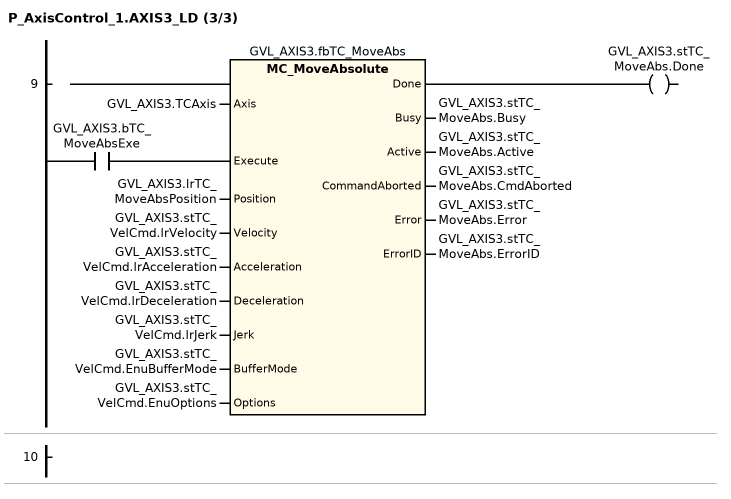
// NETWORK 9
GVL_AXIS3.fbTC_MoveAbs(
    Axis := GVL_AXIS3.TCAxis,
    Execute := GVL_AXIS3.bTC_MoveAbsExe,
    Position := GVL_AXIS3.lrTC_MoveAbsPosition,
    Velocity := GVL_AXIS3.stTC_VelCmd.lrVelocity,
    Acceleration := GVL_AXIS3.stTC_VelCmd.lrAcceleration,
    Deceleration := GVL_AXIS3.stTC_VelCmd.lrDeceleration,
    Jerk := GVL_AXIS3.stTC_VelCmd.lrJerk,
    BufferMode := GVL_AXIS3.stTC_VelCmd.EnuBufferMode,
    Options := GVL_AXIS3.stTC_VelCmd.EnuOptions,
    Busy => GVL_AXIS3.stTC_MoveAbs.Busy,
    Active => GVL_AXIS3.stTC_MoveAbs.Active,
    CommandAborted => GVL_AXIS3.stTC_MoveAbs.CmdAborted,
    Error => GVL_AXIS3.stTC_MoveAbs.Error,
    ErrorID => GVL_AXIS3.stTC_MoveAbs.ErrorID); // MC_MoveAbsolute
GVL_AXIS3.stTC_MoveAbs.Done := GVL_AXIS3.fbTC_MoveAbs.Done;

// NETWORK 10
END_METHOD

METHOD AXIS4_LD : BOOL
VAR_INPUT
END_VAR
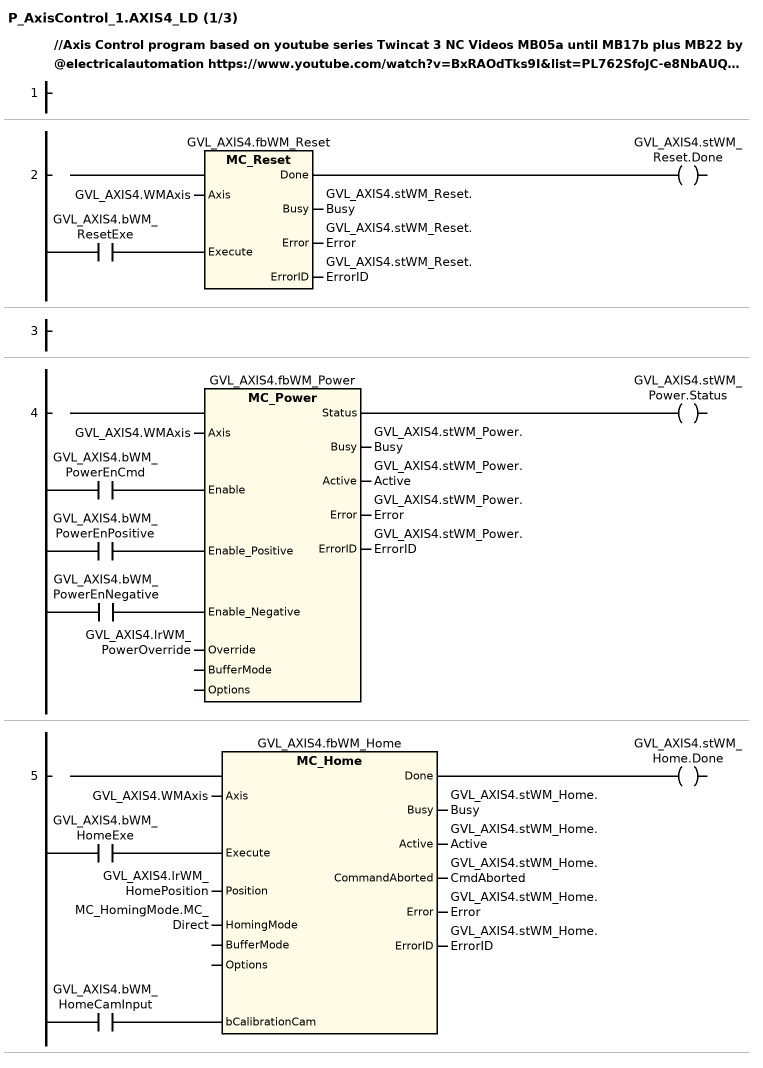
// NETWORK 1: //Axis Control program based on youtube series Twincat 3 NC Videos MB05a until MB17b plus MB22 by @electricalautomation https://www.youtube.com/watch?v=BxRAOdTks9I&list=PL762SfoJC-e8NbAUQ-H7a_TOdqrlBPCw4&index=25

// NETWORK 2
GVL_AXIS4.fbWM_Reset(
    Axis := GVL_AXIS4.WMAxis,
    Execute := GVL_AXIS4.bWM_ResetExe,
    Busy => GVL_AXIS4.stWM_Reset.Busy,
    Error => GVL_AXIS4.stWM_Reset.Error,
    ErrorID => GVL_AXIS4.stWM_Reset.ErrorID); // MC_Reset
GVL_AXIS4.stWM_Reset.Done := GVL_AXIS4.fbWM_Reset.Done;

// NETWORK 3

// NETWORK 4
GVL_AXIS4.fbWM_Power(
    Axis := GVL_AXIS4.WMAxis,
    Enable := GVL_AXIS4.bWM_PowerEnCmd,
    Enable_Positive := GVL_AXIS4.bWM_PowerEnPositive,
    Enable_Negative := GVL_AXIS4.bWM_PowerEnNegative,
    Override := GVL_AXIS4.lrWM_PowerOverride,
    Busy => GVL_AXIS4.stWM_Power.Busy,
    Active => GVL_AXIS4.stWM_Power.Active,
    Error => GVL_AXIS4.stWM_Power.Error,
    ErrorID => GVL_AXIS4.stWM_Power.ErrorID); // MC_Power
GVL_AXIS4.stWM_Power.Status := GVL_AXIS4.fbWM_Power.Status;

// NETWORK 5
GVL_AXIS4.fbWM_Home(
    Axis := GVL_AXIS4.WMAxis,
    Execute := GVL_AXIS4.bWM_HomeExe,
    Position := GVL_AXIS4.lrWM_HomePosition,
    HomingMode := MC_HomingMode.MC_Direct,
    bCalibrationCam := GVL_AXIS4.bWM_HomeCamInput,
    Busy => GVL_AXIS4.stWM_Home.Busy,
    Active => GVL_AXIS4.stWM_Home.Active,
    CommandAborted => GVL_AXIS4.stWM_Home.CmdAborted,
    Error => GVL_AXIS4.stWM_Home.Error,
    ErrorID => GVL_AXIS4.stWM_Home.ErrorID); // MC_Home
GVL_AXIS4.stWM_Home.Done := GVL_AXIS4.fbWM_Home.Done;

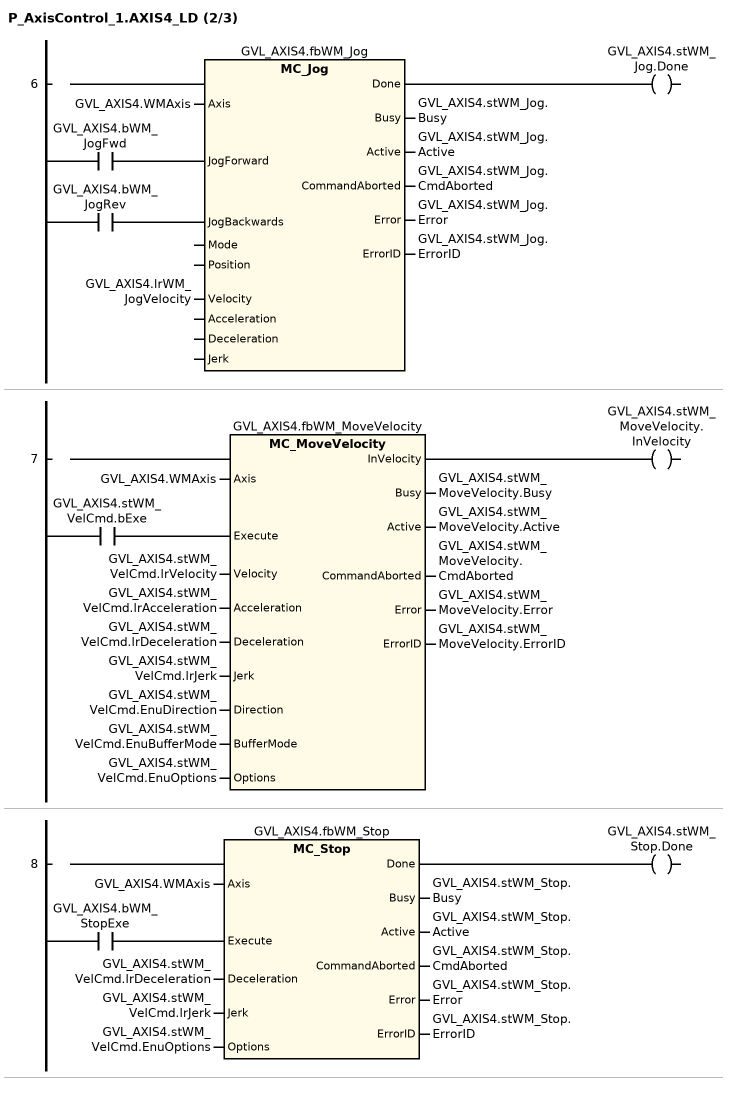
// NETWORK 6
GVL_AXIS4.fbWM_Jog(
    Axis := GVL_AXIS4.WMAxis,
    JogForward := GVL_AXIS4.bWM_JogFwd,
    JogBackwards := GVL_AXIS4.bWM_JogRev,
    Velocity := GVL_AXIS4.lrWM_JogVelocity,
    Busy => GVL_AXIS4.stWM_Jog.Busy,
    Active => GVL_AXIS4.stWM_Jog.Active,
    CommandAborted => GVL_AXIS4.stWM_Jog.CmdAborted,
    Error => GVL_AXIS4.stWM_Jog.Error,
    ErrorID => GVL_AXIS4.stWM_Jog.ErrorID); // MC_Jog
GVL_AXIS4.stWM_Jog.Done := GVL_AXIS4.fbWM_Jog.Done;

// NETWORK 7
GVL_AXIS4.fbWM_MoveVelocity(
    Axis := GVL_AXIS4.WMAxis,
    Execute := GVL_AXIS4.stWM_VelCmd.bExe,
    Velocity := GVL_AXIS4.stWM_VelCmd.lrVelocity,
    Acceleration := GVL_AXIS4.stWM_VelCmd.lrAcceleration,
    Deceleration := GVL_AXIS4.stWM_VelCmd.lrDeceleration,
    Jerk := GVL_AXIS4.stWM_VelCmd.lrJerk,
    Direction := GVL_AXIS4.stWM_VelCmd.EnuDirection,
    BufferMode := GVL_AXIS4.stWM_VelCmd.EnuBufferMode,
    Options := GVL_AXIS4.stWM_VelCmd.EnuOptions,
    Busy => GVL_AXIS4.stWM_MoveVelocity.Busy,
    Active => GVL_AXIS4.stWM_MoveVelocity.Active,
    CommandAborted => GVL_AXIS4.stWM_MoveVelocity.CmdAborted,
    Error => GVL_AXIS4.stWM_MoveVelocity.Error,
    ErrorID => GVL_AXIS4.stWM_MoveVelocity.ErrorID); // MC_MoveVelocity
GVL_AXIS4.stWM_MoveVelocity.InVelocity := GVL_AXIS4.fbWM_MoveVelocity.InVelocity;

// NETWORK 8
GVL_AXIS4.fbWM_Stop(
    Axis := GVL_AXIS4.WMAxis,
    Execute := GVL_AXIS4.bWM_StopExe,
    Deceleration := GVL_AXIS4.stWM_VelCmd.lrDeceleration,
    Jerk := GVL_AXIS4.stWM_VelCmd.lrJerk,
    Options := GVL_AXIS4.stWM_VelCmd.EnuOptions,
    Busy => GVL_AXIS4.stWM_Stop.Busy,
    Active => GVL_AXIS4.stWM_Stop.Active,
    CommandAborted => GVL_AXIS4.stWM_Stop.CmdAborted,
    Error => GVL_AXIS4.stWM_Stop.Error,
    ErrorID => GVL_AXIS4.stWM_Stop.ErrorID); // MC_Stop
GVL_AXIS4.stWM_Stop.Done := GVL_AXIS4.fbWM_Stop.Done;

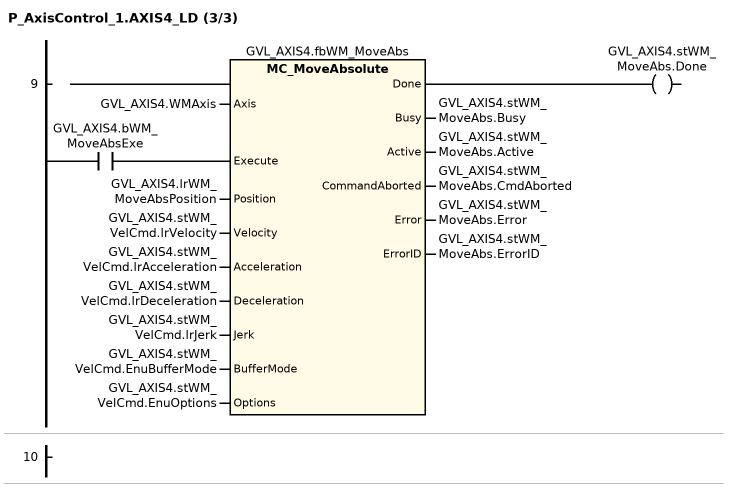
// NETWORK 9
GVL_AXIS4.fbWM_MoveAbs(
    Axis := GVL_AXIS4.WMAxis,
    Execute := GVL_AXIS4.bWM_MoveAbsExe,
    Position := GVL_AXIS4.lrWM_MoveAbsPosition,
    Velocity := GVL_AXIS4.stWM_VelCmd.lrVelocity,
    Acceleration := GVL_AXIS4.stWM_VelCmd.lrAcceleration,
    Deceleration := GVL_AXIS4.stWM_VelCmd.lrDeceleration,
    Jerk := GVL_AXIS4.stWM_VelCmd.lrJerk,
    BufferMode := GVL_AXIS4.stWM_VelCmd.EnuBufferMode,
    Options := GVL_AXIS4.stWM_VelCmd.EnuOptions,
    Busy => GVL_AXIS4.stWM_MoveAbs.Busy,
    Active => GVL_AXIS4.stWM_MoveAbs.Active,
    CommandAborted => GVL_AXIS4.stWM_MoveAbs.CmdAborted,
    Error => GVL_AXIS4.stWM_MoveAbs.Error,
    ErrorID => GVL_AXIS4.stWM_MoveAbs.ErrorID); // MC_MoveAbsolute
GVL_AXIS4.stWM_MoveAbs.Done := GVL_AXIS4.fbWM_MoveAbs.Done;

// NETWORK 10
END_METHOD

METHOD Manual_mode : BOOL
VAR_INPUT
END_VAR
AXIS1_LD();

GVL_AXIS1.bBC_ResetExe := G_Inputs.bJoystickLeftEnable;

//GVL_AXIS1.EnuMoveVelDirection := G_Sensors.MCDirectionAxis1;

GVL_AXIS1.bBC_PowerEnCmd := G_Inputs.bManualModeSelector;
GVL_AXIS1.bBC_PowerEnNegative := G_Inputs.bManualModeSelector;
GVL_AXIS1.bBC_PowerEnPositive := G_Inputs.bManualModeSelector;

IF G_Sensors.fJoystickLeftNormalizedX  > 0.01 AND G_Inputs.bJoystickLeftEnable THEN
	GVL_AXIS1.lrBC_PowerOverride := ABS(G_Sensors.fJoystickLeftNormalizedX) * 100;
	GVL_AXIS1.stBC_VelCmd.EnuDirection := MC_Positive_Direction;
	GVL_AXIS1.stBC_VelCmd.bExe := TRUE;
ELSIF G_Sensors.fJoystickLeftNormalizedX < 0.01 AND G_Inputs.bJoystickLeftEnable THEN
	GVL_AXIS1.lrBC_PowerOverride := ABS(G_Sensors.fJoystickLeftNormalizedX) * 100;
	GVL_AXIS1.stBC_VelCmd.EnuDirection := MC_Negative_Direction;
	GVL_AXIS1.stBC_VelCmd.bExe := TRUE;
END_IF
END_METHOD

END_PROGRAM

// ---- INPUTS/P_Inputs.TcPOU
PROGRAM P_Inputs
VAR
	fbJoystickLeftVert 					: FB_JoystickInputScaling;
	fbJoystickLeftHor 					: FB_JoystickInputScaling;
	
	fbJoystickRightVert 				: FB_JoystickInputScaling;
	fbJoystickRightHor 					: FB_JoystickInputScaling;
	
	bEnableJoystick : BOOL;
		
END_VAR

bEnableJoystick := NOT(P_StablePlatform.bManualMode);

fbJoystickLeftVert(
	bEnable := bEnableJoystick,
	nRawInput := G_Inputs.stJoyLY.nValue,
	stJoystickInputScaling := G_ScalingParameters.stParam.stJoystickInputScalingLeftY,
	fNormalizedOutput => G_Sensors.fJoystickLeftNormalizedY
);

IF G_Sensors.fJoystickLeftNormalizedY < 0 THEN
	G_Sensors.MCDirectionAxis3 := MC_Negative_Direction;
ELSIF G_Sensors.fJoystickLeftNormalizedY > 0 THEN
	G_Sensors.MCDirectionAxis3 := MC_Positive_Direction;	
END_IF

fbJoystickLeftHor(
	bEnable := bEnableJoystick,
	nRawInput := G_Inputs.stJoyLX.nValue,
	stJoystickInputScaling := G_ScalingParameters.stParam.stJoystickInputScalingLeftX,
	fNormalizedOutput => G_Sensors.fJoystickLeftNormalizedX
);

IF G_Sensors.fJoystickLeftNormalizedX < 0 THEN
	G_Sensors.MCDirectionAxis1 := MC_Positive_Direction;
ELSIF G_Sensors.fJoystickLeftNormalizedX > 0 THEN
	G_Sensors.MCDirectionAxis1 := MC_Negative_Direction;	
END_IF


fbJoystickRightVert(
	bEnable := bEnableJoystick,
	nRawInput := G_Inputs.stJoyRY.nValue,
	stJoystickInputScaling := G_ScalingParameters.stParam.stJoystickInputScalingRightY,
	fNormalizedOutput => G_Sensors.fJoystickRightNormalizedY
);

IF G_Sensors.fJoystickRightNormalizedY < 0 THEN
	G_Sensors.MCDirectionAxis4 := MC_Negative_Direction;
ELSIF G_Sensors.fJoystickRightNormalizedY > 0 THEN
	G_Sensors.MCDirectionAxis4 := MC_Positive_Direction;	
END_IF



fbJoystickRightHor(
	bEnable := bEnableJoystick,
	nRawInput := G_Inputs.stJoyRX.nValue,
	stJoystickInputScaling := G_ScalingParameters.stParam.stJoystickInputScalingRightX,
	fNormalizedOutput => G_Sensors.fJoystickRightNormalizedX
);

IF G_Sensors.fJoystickRightNormalizedX < 0 THEN
	G_Sensors.MCDirectionAxis2 := MC_Positive_Direction;
ELSIF G_Sensors.fJoystickRightNormalizedX > 0 THEN
	G_Sensors.MCDirectionAxis2 := MC_Negative_Direction;	
END_IF

END_PROGRAM

// ---- StablePlatform/P_StablePlatform.TcPOU
PROGRAM P_StablePlatform
VAR
	fbpA 		: FB_AnalogInputScaling;
	fbpB 		: FB_AnalogInputScaling;
	fbpS 	 	: FB_AnalogInputScaling;
	fSVFeedback : FB_AnalogInputScaling;
	fbPistonPos	: FB_AnalogInputScaling_1;
	fbPistonVel	: FB_AnalogInputScaling_1;
	fbJoystick  : FB_JoystickInputScaling;
	fbSVOutput 	: FB_ValveOutput;
	bManualMode : BOOL;
END_VAR

// Inputs
fbpA(
	nRawInput := G_StablePlatformIO.npA,
	stAnalogInputScaling := G_StablePlatformParameters.stPressureSensorScaling400bar,
	fOutput => G_StablePlatformScaledIO.bpA
);

fbpB(
	nRawInput := G_StablePlatformIO.npB,
	stAnalogInputScaling := G_StablePlatformParameters.stPressureSensorScaling400bar,
	fOutput => G_StablePlatformScaledIO.bpB
);

fbpS(
	nRawInput := G_StablePlatformIO.npS,
	stAnalogInputScaling := G_StablePlatformParameters.stPressureSensorScaling400bar,
	fOutput => G_StablePlatformScaledIO.bpS
);

fSVFeedback(
	nRawInput := G_StablePlatformIO.nSVFeedback,
	stAnalogInputScaling := G_StablePlatformParameters.stSVFeedbackScaling,
	fOutput => G_StablePlatformScaledIO.fSVFeedback
);


fbJoystick(
	bEnable := bManualMode,
	nRawInput := G_Inputs.stJoyLX.nValue,
	stJoystickInputScaling := G_StablePlatformParameters.stJoystickInputScalingX,
	fNormalizedOutput => G_StablePlatformScaledIO.fJoystickNormalizedX
);

// Outputs
fbSVOutput(
	bEnable := G_Inputs.bJoystickLeftEnable AND bManualMode,
	bDeadBandCompOn := FALSE,
	stValveDeadBand := G_StablePlatformParameters.stSVValveDeadBand,
	fNormalizedInput := -G_StablePlatformScaledIO.fJoystickNormalizedX,
	nOutput => G_StablePlatformIO.nSVControlSignal
);

G_StablePlatformIO.bSVEnable := bManualMode AND G_StablePlatformIO.bEMG_OK;

fbPistonPos(
	nRawInput := G_StablePlatformIO.nPistonPosition,
	stAnalogInputScaling := G_StablePlatformParameters.stPistonPos,
	fOutput => G_StablePlatformScaledIO.fPistonPosition
);


fbPistonVel(
	nRawInput := G_StablePlatformIO.nPistonVelocity,
	stAnalogInputScaling := G_StablePlatformParameters.stPistonVel,
	fOutput => G_StablePlatformScaledIO.fPistonVelocity
);


G_StablePlatformParameters.fPlatformAngle := fPlatformAngleTheta1(fStroke:=G_StablePlatformScaledIO.fPistonPosition);

END_PROGRAM

// ---- StablePlatform/Function Blocks/FB_ValveOutput.TcPOU
FUNCTION_BLOCK FB_ValveOutput
VAR_INPUT
	bEnable 			: BOOL;
	bDeadBandCompOn 	: BOOL;
	stValveDeadBand 	: ST_ValveDeadBand;
	fNormalizedInput 	: LREAL;
END_VAR
VAR_OUTPUT
	bEnableValveOutput : BOOL;
	nOutput : INT; 
END_VAR
VAR
	nOffset 	: INT := 16383;
	nMaxValue	: INT := 32767;
	nMinValue 	: INT := 0;
	nTempOutput : INT;
END_VAR

IF	bDeadBandCompOn THEN
	IF fNormalizedInput > 0.0 THEN
		nTempOutput := LREAL_TO_INT(ABS(fNormalizedInput*(stValveDeadBand.fPosMax - stValveDeadBand.fPosMin) + stValveDeadBand.fPosMin));
	ELSIF fNormalizedInput < 0.0 THEN
		nTempOutput := LREAL_TO_INT(ABS(fNormalizedInput*(stValveDeadBand.fNegMax - stValveDeadBand.fNegMin) - stValveDeadBand.fNegMin));
	ELSE
		nTempOutput := nOffset;
	END_IF
ELSE
	IF fNormalizedInput > 0.0 THEN
		nTempOutput := LREAL_TO_INT(ABS(fNormalizedInput*(32767.0 - 16383.0) + 16383.0));
	ELSIF fNormalizedInput < 0.0 THEN
		nTempOutput := LREAL_TO_INT(ABS(fNormalizedInput*(0 - 16383.0) - 16383.0));
	ELSE
		nTempOutput := nOffset;
	END_IF	
END_IF	

IF bEnable THEN
	nOutput := LIMIT(nMinValue, nTempOutput, nMaxValue);
	bEnableValveOutput := TRUE; 
ELSE 	
	nOutput := nOffset;
	bEnableValveOutput := FALSE;	
END_IF

END_FUNCTION_BLOCK

// ---- StablePlatform/fPlatformAngleTheta1.TcPOU
FUNCTION fPlatformAngleTheta1 : LREAL
VAR_INPUT
	fStroke : LREAL;
	
END_VAR
VAR_OUTPUT
	fPlatformAngle : LREAL;
END_VAR
VAR
	fAngleBeta		: LREAL;
	fCylinderLength	: LREAL;
	fMinLength 		: LREAL; 
END_VAR

fMinLength := G_StablePlatformParameters.fMinLengthPlatformCylinder;

fCylinderLength := fStroke + fMinLength;

fAngleBeta := ACOS((G_StablePlatformParameters.fLengthA*G_StablePlatformParameters.fLengthA +  G_StablePlatformParameters.fLengthC*G_StablePlatformParameters.fLengthC - fCylinderLength*fCylinderLength) / (2 * G_StablePlatformParameters.fLengthA * G_StablePlatformParameters.fLengthC));

fPlatformAngle := -(fAngleBeta - G_StablePlatformParameters.fOffsetAngleRad);

END_FUNCTION

// ---- MACHINE CONTROL/KinematicFunctions2d/FB_Forward.TcPOU
FUNCTION_BLOCK FB_Forward
VAR_INPUT
	fTheta1: LREAL;
	fStrokeActuatorMain: LREAL;
	fStrokeActuatorKnuckle: LREAL;
END_VAR
VAR_OUTPUT
	x: LREAL;
	y: LREAL;
	fTheta3: LREAL;
	fTheta4: LREAL;
END_VAR
VAR
	x_tmp: LREAL;
	x_tmp_0: LREAL;
END_VAR


(* MATLAB Function: '<Root>/Forward kinematics actuator strokes' *)
(* Platform constants *)
(* MATLAB Function 'Forward kinematics actuator strokes': '<S1>:1' *)
(* '<S1>:1:4' fHeightPlatform = 1.402; *)
(* '<S1>:1:5' fHeightPlatformKing = 0.09; *)
(* '<S1>:1:6' fLengthPlatform = 1.30; *)
(* Crane and platform dimensions *)
(* Crane constant parameters *)
(* '<S1>:1:11' fHeightKingSlew             = 0.623; *)
(* '<S1>:1:12' fHeightSlewTop              = 0.711; *)
(* '<S1>:1:13' fLengthMainArm			    = 1.5; *)
(* '<S1>:1:14' fLengthKnuckleArm		    = 1.158; *)
(* '<S1>:1:16' fLengthAMain				= 0.614; *)
(* '<S1>:1:17' fLengthBMain				= 0.571; *)
(* '<S1>:1:18' fMinLengthActuatorMain		= 0.692; *)
(* '<S1>:1:19' fMaxStrokeActuatorMain		= 0.320; *)
(* '<S1>:1:21' fOffsetAngleDegMainAct		= 62.1; *)
(* '<S1>:1:22' fOffsetAngleRadMainAct		= deg2rad(fOffsetAngleDegMainAct); *)
(* '<S1>:1:24' fLengthAKnuckle				= 0.767; *)
(* '<S1>:1:25' fLengthBKnuckle				= 0.184; *)
(* '<S1>:1:26' fMinLengthActuatorKnuckle	= 0.627; *)
(* '<S1>:1:27' fMaxStrokeActuatorKnuckle	= 0.260; *)
(* '<S1>:1:29' fOffsetAngleDegKnuckleAct	= 86.3; *)
(* '<S1>:1:30' fOffsetAngleRadKnuckleAct	= deg2rad(fOffsetAngleDegKnuckleAct); *)
(* Calculating angles for main arm *)
(* '<S1>:1:33' fLengthActuatorMain = fStrokeActuatorMain + fMinLengthActuatorMain; *)
(* '<S1>:1:35' fAngleMainArmAct = acos((fLengthBMain^2 + fLengthAMain^2 - fLengthActuatorMain^2) / (2 * fLengthBMain * fLengthAMain)); *)
(* '<S1>:1:37' fTheta3 = fAngleMainArmAct - fOffsetAngleRadMainAct; *)
fTheta3 := ACOS((0.70303699999999991 - ((fStrokeActuatorMain + 0.692) * (fStrokeActuatorMain + 0.692))) / 0.70118799999999992) - 1.0838494654884787;
(* Calculating angles for knuckle arm *)
(* '<S1>:1:40' fLengthActuatorKnuckle = fStrokeActuatorKnuckle + fMinLengthActuatorKnuckle; *)
(* '<S1>:1:42' fAngleKnuckleArmAct = acos((fLengthBKnuckle^2 + fLengthAKnuckle^2 - fLengthActuatorKnuckle^2) / (2 * fLengthBKnuckle * fLengthAKnuckle)); *)
(* '<S1>:1:44' fTheta4 = fAngleKnuckleArmAct - fOffsetAngleRadKnuckleAct; *)
fTheta4 := ACOS((0.62214500000000006 - ((fStrokeActuatorKnuckle + 0.627) * (fStrokeActuatorKnuckle + 0.627))) / 0.282256) - 1.5062191444711064;

(* fAngleMainArmAct			= fTheta3deg + fOffsetAngleDegMainAct; *)
(* fAngleKnuckleArmAct         = fTheta4deg + fOffsetAngleDegKnuckleAct; *)

(* fLengthActuatorMain         = sqrt(fLengthAMain^2 + fLengthBMain^2 -(2*fLengthAMain*fLengthBMain*cosd(fAngleMainArmAct))); *)
(* fStrokeActuatorMain         = fLengthActuatorMain - fMinLengthActuatorMain; *)
(* if fStrokeActuatorMain < 0 *)
(* fStrokeActuatorMain = 0; *)
(* elseif fStrokeActuatorMain > fMaxStrokeActuatorMain *)
(* fMaxStrokeActuatorMain = fMaxStrokeActuatorMain; *)
(* end *)

(* fLengthActuatorKnuckle         = sqrt(fLengthAKnuckle^2 + fLengthBKnuckle^2 -(2*fLengthAKnuckle*fLengthBKnuckle*cosd(fAngleKnuckleArmAct))); *)
(* fStrokeActuatorKnuckle         = fLengthActuatorKnuckle - fMinLengthActuatorKnuckle; *)

(* if fStrokeActuatorKnuckle < 0 *)
(* fStrokeActuatorKnuckle = 0; *)
(* elseif fStrokeActuatorKnuckle > fMaxStrokeActuatorKnuckle *)
(* fMaxStrokeActuatorKnuckle = fMaxStrokeActuatorKnuckle; *)
(* end *)
(* '<S1>:1:71' fHeightMain                 = fHeightPlatformKing + fHeightKingSlew + fHeightSlewTop; *)
(* x = fLengthPlatform*cos(fTheta1) + fHeightMain*cos(fTheta1 + pi/2) + fLengthMainArm*cos(fTheta1 + fTheta3) + fLengthKnuckleArm * cos (fTheta1 + fTheta3 + fTheta4 - pi/2); *)
(* y = fHeightPlatform + fLengthPlatform*sin(fTheta1) + fHeightMain * sin(fTheta1 + pi/2) + fLengthMainArm *sin(fTheta1 + fTheta3) + fLengthKnuckleArm*sin(fTheta1 + fTheta3 + fTheta4 - pi/2); *)
(* '<S1>:1:76' x = fLengthPlatform*cos(fTheta1) + fHeightMain*cos(fTheta1 + pi/2) + fLengthMainArm*cos(fTheta1 + fTheta3) + fLengthKnuckleArm * cos (fTheta1 + fTheta3 + fTheta4 - pi/2); *)
(* '<S1>:1:77' y = fHeightPlatform + fLengthPlatform*sin(fTheta1) + fHeightMain * sin(fTheta1 + pi/2) + fLengthMainArm *sin(fTheta1 + fTheta3) + fLengthKnuckleArm*sin(fTheta1 + fTheta3 + fTheta4 - pi/2); *)
x_tmp := fTheta1 + fTheta3;
x_tmp_0 := (x_tmp + fTheta4) - 1.5707963267948966;
(* Outport: '<Root>/x' incorporates:
 *  MATLAB Function: '<Root>/Forward kinematics actuator strokes' *)
x := (((COS(fTheta1 + 1.5707963267948966) * 1.424) + (1.3 * COS(fTheta1))) + (COS(x_tmp) * 1.5)) + (COS(x_tmp_0) * 1.158);
(* Outport: '<Root>/y' incorporates:
 *  MATLAB Function: '<Root>/Forward kinematics actuator strokes' *)
y := ((((1.3 * SIN(fTheta1)) + 1.402) + (SIN(fTheta1 + 1.5707963267948966) * 1.424)) + (SIN(x_tmp) * 1.5)) + (SIN(x_tmp_0) * 1.158);

END_FUNCTION_BLOCK

// ---- StablePlatform/Function Blocks/FB_JoystickInputScaling_1.TcPOU
FUNCTION_BLOCK FB_JoystickInputScaling_1
VAR_INPUT
	bEnable 				: BOOL;
	nRawInput 				: INT;
	stJoystickInputScaling  : ST_JoystickInputScaling;
END_VAR
VAR_OUTPUT
	fNormalizedOutput 		: LREAL;
END_VAR
VAR
	fRawInput 				: LREAL;
	fTempInput 				: LREAL;
	fTempOutput 			: LREAL;
END_VAR

fRawInput := INT_TO_LREAL(nRawInput);

fTempInput := fRawInput - stJoystickInputScaling.fNeutralInputValue;

IF fTempInput > stJoystickInputScaling.fNeutralDeadband THEN
	fTempOutput := fTempInput/(stJoystickInputScaling.fMaxInputValue - stJoystickInputScaling.fNeutralInputValue);
ELSIF fTempInput < -stJoystickInputScaling.fNeutralDeadband THEN	
	fTempOutput := fTempInput/(stJoystickInputScaling.fNeutralInputValue - stJoystickInputScaling.fMinInputValue);
ELSE
	fTempOutput := 0.0;
END_IF

IF NOT(bEnable) THEN
	fNormalizedOutput := 0.0;
ELSE
	fNormalizedOutput := LIMIT(stJoystickInputScaling.fMinOutputValue, fTempOutput, stJoystickInputScaling.fMaxOutputValue);
END_IF

END_FUNCTION_BLOCK

// ---- GlobalTextList.TcGTLO
TEXTLIST GlobalTextList
  24 = '%f'
  695 = '%f Cylinder Position [m]'
  963 = '%f Cylinder Velocity [m/s]'
  798 = '24VDC PowerRefresh'
  519 = 'AcknowAledge'
  820 = 'Acknowledge'
  23 = 'Active'
  890 = 'Drive STO'
  810 = 'EMG Stop'
  418 = 'Enable'
  942 = 'Group'
  463 = 'Group                                   Run/Stop'
  914 = 'Group Run/Stop'
  708 = 'GroupBox'
  107 = 'PowerRefresh'
  181 = 'Restart'
  267 = 'Run/Stop'
  114 = 'Stable Platform'
  488 = 'TwinSAFE'
END_TEXTLIST

// ---- HMI/HMI.TcVIS
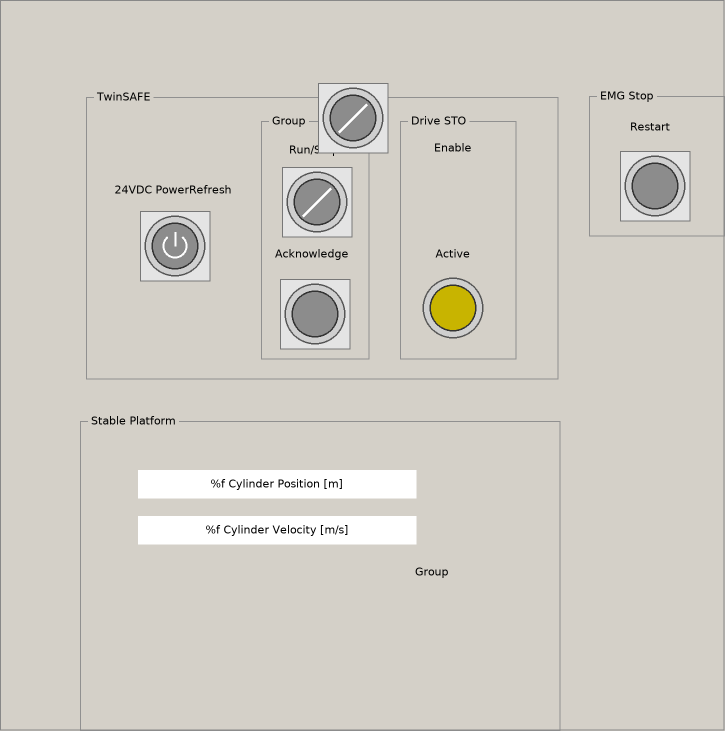
VISUALIZATION HMI  // 725x731
    GroupBox (86,89 472x290), "TwinSAFE"
        Label (268,468 156x30), "Group"
        Label (150,46 156x30), "Run/Stop"
        Label (148,150 156x30), "Acknowledge"
        GroupBox (175,24 108x246), "Group"
            RotarySwitch (21,54 70x70), variable: GVL_Safety_AXIS4.TwinSafeGroupRunStop, behaviour: TOGGLE, style: Switch-RotarySwitch-Gray
            PushSwitch (19,166 70x70), variable: GVL_Safety_AXIS4.TwinSafeGroupComErrAck, behaviour: TAP, style: Switch-PushSwitch-Gray
        Lamp1 (170,918 70x70), variable: GVL_Safety_AXIS4.ChA_STO_Active, style: Lamp-Lamp1-Yellow
        GroupBox (314,24 116x246), "Drive STO"
            RotarySwitch (-82,-30 70x70), behaviour: TOGGLE, style: Switch-RotarySwitch-Gray
            Lamp1 (18,160 70x70), variable: GVL_Safety_AXIS4.ChA_STO_Active, style: Lamp-Lamp1-Yellow
        Label (292,44 150x30), "Enable"
        Label (292,150 150x30), "Active"
        PowerSwitch (54,122 70x70), variable: GVL_Safety_AXIS4.bWinchMotor24vDisable, behaviour: TAP, style: Switch-PowerSwitch-Gray
        Label (12,86 150x30), "24VDC PowerRefresh"
    GroupBox (80,413 480x318), "Stable Platform"
        Textfield (57,56 280x30), "%f Cylinder Position [m]", text variable: G_StablePlatformScaledIO.fPistonPosition
        Textfield (57,102 280x30), "%f Cylinder Velocity [m/s]", text variable: G_StablePlatformScaledIO.fPistonVelocity
    GroupBox (589,88 136x148), "EMG Stop"
        PushSwitch (31,63 70x70), variable: GVL_Safety_AXIS4.EMGRestart, behaviour: TAP, style: Switch-PushSwitch-Gray
    Label (575,112 150x30), "Restart"
END_VISUALIZATION
